// ====== process functions if enabled ======
	// ***** Set Delayed inputs and time elapsed ****
		FB_delIStatus(	IN:= bFcoInputActive,
						PT:= tDelay , 
						Q=> bFcoDelay , 
						ET=> TetInputActive 
					  ); // Generate delayed input status from push button input status
	// ***** Edge triggers *****
		FB_feIStatus(CLK:= Istatus , Q=> bFeStatus ); // generate falling edge pulse on pushbutton input
		FB_reIStatus (Clk := Istatus , Q => bReStatus); // Generate rising edge from push button input signal

END_FUNCTION_BLOCK

// Buttons/Functions/FB_DevPushButton
FUNCTION_BLOCK PUBLIC FB_DevPushButton EXTENDS Fb_DevDigitalInputFunctions
VAR_INPUT
END_VAR
VAR_OUTPUT
END_VAR
VAR
END_VAR

// set device type
IF eDevType = E_Devices.Undefined THEN 
	eDevType := E_Devices.DigitalSensor ;
END_IF

SUPER^();

END_FUNCTION_BLOCK

// Encoders/FunctionBlocks/FB_EncoderBase
FUNCTION_BLOCK PUBLIC FB_EncoderBase
VAR_INPUT
	nCfgUnitsPerPulse	: LREAL := 1	; // Scale factor for output [units/pulse]
	nCfgOffset			: LREAL := 0	; // Offset for output
	
	bIcfInverted		: BOOL	:= FALSE; // Invert output position = standard false  
END_VAR
VAR_OUTPUT
	nOutPosition		: LREAL	:= 0	; // Scaled position output
	nOutRaw				: UDINT := 0	; // Raw output value	 
	nVelocity			: LREAL	:= 0 	; // Velocity [units/sec]
END_VAR
VAR
END_VAR

METHOD PUBLIC FastTask : BOOL
VAR_INPUT
END_VAR
END_METHOD

END_FUNCTION_BLOCK

// Encoders/FunctionBlocks/FB_EncoderInput
FUNCTION_BLOCK FB_EncoderInput EXTENDS FB_EncoderBase
VAR_INPUT
END_VAR
VAR_OUTPUT
END_VAR
VAR
	iEncoderSignal AT%I*: UDINT ;
	
	nScaledValue		: LREAL ; // Only scaled value for internal use
	nValueWithOffset	: LREAL ; // scaled value with added offset
END_VAR

// ====== Scale Output value ======
	nScaledValue := UDINT_TO_LREAL(iEncoderSignal) * nCfgUnitsPerPulse ;

// ====== Invert ======
	IF bIcfInverted THEN 
		nScaledValue := nScaledValue * -1;
	END_IF
	
// ====== Add offset ======= 
	nValueWithOffset := nScaledValue + nCfgOffset ;

// ====== Set Outputs =======
	nOutPosition 	:= nValueWithOffset ;
	nOutRaw			:= iEncoderSignal	;

METHOD PUBLIC FastTask : BOOL
VAR_INPUT
END_VAR
END_METHOD

END_FUNCTION_BLOCK

// HardwareDiagnostics/FB_ELModuleDiag
FUNCTION_BLOCK PUBLIC FB_ELModuleDiag
VAR_INPUT
END_VAR
VAR_OUTPUT
	bError 	:	BOOL ; // Module is in error
	sErrorDiscription : STRING ; // module error discription 
END_VAR
VAR
END_VAR

END_FUNCTION_BLOCK

// Outputs/AnalogOutputs/FB_DevAnalogOutputScaled
FUNCTION_BLOCK FB_DevAnalogOutputScaled EXTENDS FB_DevAnalogOutput
VAR_INPUT
END_VAR
VAR_OUTPUT
END_VAR
VAR
	fGainFactor 	: LREAL:= 32767	;
END_VAR

SUPER^();

METHOD INTERNAL ExecSetFeedback : BOOL
VAR_INPUT
END_VAR
// Set feedback 
fOutputValue := qnHwOut ;
END_METHOD

METHOD INTERNAL ExecSetOutput : BOOL
VAR_INPUT
END_VAR
// Set Output to physical device
IF bEnable OR bCmdManual THEN 
	qnHwOut := LREAL_TO_INT(fCmdValue * fGainFactor) ;
	qnHwOut := LIMIT(nLimitMin, qnHwOut, nLimitMax) ; 
ELSE 
	fCmdValue := 0 ; 
END_IF
END_METHOD

METHOD PUBLIC SetScaling : BOOL 
VAR_INPUT
	fMaxValue	: LREAL ; 		// Maximum input value after scaling, e.g. 100% (mandatory input)  
END_VAR
// calculate gain 
fGainFactor := nLimitMax / fMaxValue ;
END_METHOD

END_FUNCTION_BLOCK

// Sensors/AnalogInput/FunctionBlocks/FB_DevAnalogInAutoCalibrate
FUNCTION_BLOCK PUBLIC FB_DevAnalogInAutoCalibrate EXTENDS FB_DevAnalogInputScaled
VAR_INPUT
END_VAR
VAR_OUTPUT
END_VAR
VAR
END_VAR

SUPER^();

METHOD PUBLIC CmdCalibrateNull : BOOL
VAR_INPUT
END_VAR
// set offset to calibrate to null
nOfset := - inHwInput ;
END_METHOD

METHOD PUBLIC CmdCalilbrateValue : BOOL // calibrate gain factor to actual value (warning calibrate to null before calibrating to value)
VAR_INPUT
	fCalibrationValue	: LREAL ; // Active input value to sensor (calibration setpoint)
END_VAR
// set gain from current value
fGainFactor := INT_TO_LREAL(inHwInput + nOfset) / fCalibrationValue ;
END_METHOD

END_FUNCTION_BLOCK

// Sensors/AnalogInput/FunctionBlocks/FB_DevAnalogInputScaled
FUNCTION_BLOCK PUBLIC FB_DevAnalogInputScaled EXTENDS FB_DevAnalogInput
VAR_INPUT
END_VAR
VAR_OUTPUT
END_VAR
VAR
	fGainFactor 	: LREAL	:= 1	;
	nOfset			: INT	:= 0	;
END_VAR

SUPER^();

METHOD ExecSetFeedback : BOOL
VAR
	nCalibValue	: INT ; 
END_VAR
// Offset 
IF bCmdSimulate THEN 
	nCalibValue := fSimValue + nOfset ;
ELSE
	nCalibValue := inHwInput + nOfset ;
END_IF

fValue := INT_TO_LREAL(nCalibValue) / fGainFactor;
END_METHOD

METHOD PUBLIC SetScaling : BOOL 
VAR_INPUT
	fMaxValue	: LREAL ; 	// Maximum input value after scaling, e.g. 100%, 0 = no scaling (gain = hardware limit / fMaxValue)  
	fOfset		: LREAL ;	// offset value (fvalue = (gain * hwvalue) + fOfset)
END_VAR
// calculate gain 
IF fMaxValue =0 THEN 
	fGainFactor := 1 ;
ELSE 
	fGainFactor := nLimitMax / fMaxValue ;
END_IF

nOfset := LREAL_TO_INT(fOfset * fGainFactor) ;
END_METHOD

END_FUNCTION_BLOCK

// Sensors/AnalogInput/FunctionBlocks/FB_DevHDAnalogInAutoCalibrate
FUNCTION_BLOCK PUBLIC FB_DevHDAnalogInAutoCalibrate EXTENDS FB_DevHDAnalogInputScaled
VAR_INPUT
END_VAR
VAR_OUTPUT
END_VAR
VAR
END_VAR

SUPER^();

METHOD PUBLIC CmdCalibrateNull : BOOL
VAR_INPUT
END_VAR
// set offset to calibrate to null
nOfset := - inHwInput ;
END_METHOD

METHOD PUBLIC CmdCalilbrateValue : BOOL // calibrate gain factor to actual value (warning calibrate to null before calibrating to value)
VAR_INPUT
	fCalibrationValue	: LREAL ; // Active input value to sensor (calibration setpoint)
END_VAR
// set gain from current value
fGainFactor := DINT_TO_LREAL(inHwInput + nOfset) / fCalibrationValue ;
END_METHOD

END_FUNCTION_BLOCK

// Sensors/AnalogInput/FunctionBlocks/FB_DevHDAnalogInputScaled
FUNCTION_BLOCK PUBLIC FB_DevHDAnalogInputScaled EXTENDS FB_DevHDAnalogInput
VAR_INPUT
END_VAR
VAR_OUTPUT
END_VAR
VAR
	fGainFactor 	: LREAL	:= 1	;
	nOfset			: DINT	:= 0	;
END_VAR

SUPER^();

METHOD ExecSetFeedback : BOOL
VAR
	nCalibValue	: DINT ; 
END_VAR
// Offset 
IF bCmdSimulate THEN 
	nCalibValue := fSimValue + nOfset ;
ELSE
	nCalibValue := inHwInput + nOfset ;
END_IF

fValue := DINT_TO_LREAL(nCalibValue) / fGainFactor;
END_METHOD

METHOD PUBLIC SetScaling : BOOL 
VAR_INPUT
	fMaxValue	: LREAL ; 	// Maximum input value after scaling, e.g. 100%, 0 = no scaling (gain = hardware limit / fMaxValue)  
	fOfset		: LREAL ;	// offset value (fvalue = (gain * hwvalue) + fOfset)
END_VAR
// calculate gain 
IF fMaxValue =0 THEN 
	fGainFactor := 1 ;
ELSE 
	fGainFactor := nLimitMax / fMaxValue ;
END_IF

nOfset := LREAL_TO_DINT(fOfset * fGainFactor) ;

SetScaling := TRUE ;
END_METHOD

END_FUNCTION_BLOCK

// Sensors/AnalogInput/FunctionBlocks/FB_DevHDAnalogInput
FUNCTION_BLOCK PUBLIC FB_DevHDAnalogInput EXTENDS FB_DevBase
VAR_INPUT
	bCmdSimulate	: BOOL 	:= FALSE ;// Simulate sensor Input 
	fSimValue		: DINT	:= 0 ;// Simulated sensor state
END_VAR
VAR_OUTPUT
	fValue	: LREAL := 0 ; // Analog input value (LREAL)
END_VAR
VAR
	nLimitMin		: DINT := Utilities_Library.GVL_FixedValues.nDINTMINVALUE	; // Initial value is set to integer minimum value for use with normal def analog inputs 
	nLimitMax 		: DINT := Utilities_Library.GVL_FixedValues.nDINTMAXVALUE 	; // Initial value is set to integer minimum value for use with high def analog inputs
	inHwInput AT%I* : DINT ; // Hardware connection
END_VAR

// Set device type
eDevType := E_Devices.AnalogSensor ;

// Call base function
SUPER^();

// set feedback
ExecSetFeedback();

METHOD ExecSetFeedback : BOOL
VAR_INPUT
END_VAR
IF bCmdSimulate THEN 
	fValue := fSimValue ;
ELSE
	fValue := DINT_TO_LREAL(inHwInput);
END_IF
END_METHOD

END_FUNCTION_BLOCK

// Sensors/FootPedals/FunctionBlocks/FB_EfkaEB301A_FootPedal
FUNCTION_BLOCK PUBLIC FB_EfkaEB301A_FootPedal
VAR_INPUT
	bEnable : BOOL := TRUE ;
END_VAR
VAR_OUTPUT
	ePedalInputStep		: E_FootpedalPos	:= 0 ;
	bRTrigtoReverse1 	: BOOL := FALSE ; // rising edge trigger when pedal moves from 0 to -1 or Idle to reverse 1 
	bRTrigtoReverse2 	: BOOL := FALSE ; // rising edge trigger when pedal moves from 1 to -2 or reverse 1 to reverse 2 
	bRTrigtoForward1 	: BOOL := FALSE ; // rising edge trigger when pedal moves from 0 to 1 or idle to forward 1 
	bRTrigtoForward2 	: BOOL := FALSE ; // rising edge trigger when pedal moves from 0 to 1 or forward to forward 2 
END_VAR
VAR
	// ===== greycode switches from footpedal =====
	I_GreyCodeA AT%I* : BOOL	; // Greycode input a from foot pedal 
	I_GreyCodeB AT%I* : BOOL	; // Greycode input a from foot pedal 
	I_GreyCodeC AT%I* : BOOL	; // Greycode input a from foot pedal 
	I_GreyCodeD AT%I* : BOOL	; // Greycode input a from foot pedal 
	nGreyCodetotal	: BYTE ; // all greycode switches combined
	// ==== decimal value =====
	ePreviousPedalInput	: E_FootpedalPos	:= 0 ;
END_VAR

// ===== Read input from pedal =====
ACT_ConvertGreycode();

// ===== Create edge flanks for functions =====
ACT_CreateEdges();

ACTION ACT_ConvertGreycode:
// ===== Combine greycode sensors =====
nGreyCodetotal.0 := I_GreyCodeA ;
nGreyCodetotal.1 := I_GreyCodeB ;
nGreyCodetotal.2 := I_GreyCodeB ;
nGreyCodetotal.3 := I_GreyCodeC ;

// ==== Convert greycode decimal to speed steps =====
// this only makes sense in EFKA world but anyway let's convert it to our own sense
CASE nGreyCodetotal OF 
	12: ePedalInputStep := E_FootpedalPos.eReverse1	;
	14: ePedalInputStep := E_FootpedalPos.eReverse2	;
	15: ePedalInputStep := E_FootpedalPos.eIdle		;
	13: ePedalInputStep := E_FootpedalPos.eForward1	;
	09: ePedalInputStep := E_FootpedalPos.eForward2	;
 	08: ePedalInputStep := E_FootpedalPos.eForward3	;
	10: ePedalInputStep := E_FootpedalPos.eForward4	;
	11: ePedalInputStep := E_FootpedalPos.eForward5	;
	03:	ePedalInputStep := E_FootpedalPos.eForward6	;
	02:	ePedalInputStep := E_FootpedalPos.eForward7	;
	00: ePedalInputStep := E_FootpedalPos.eForward8	;
	01: ePedalInputStep := E_FootpedalPos.eForward9	;
	05: ePedalInputStep := E_FootpedalPos.eForward10	;
	04: ePedalInputStep := E_FootpedalPos.eForward11	;
	06: ePedalInputStep := E_FootpedalPos.eForward12 	;
	07: ePedalInputStep := E_FootpedalPos.eForward13	;
	ELSE
		ePedalInputStep := E_FootpedalPos.eFalse 		;
END_CASE
END_ACTION

ACTION ACT_CreateEdges:
// ===== create edges on which functions can be triggerd =====
CASE ePedalInputStep OF
	E_FootpedalPos.eReverse2:
		bRTrigtoReverse2 := ePreviousPedalInput = E_FootpedalPos.eReverse1 ;
	E_FootpedalPos.eReverse1:
		bRTrigtoReverse1 := ePreviousPedalInput = E_FootpedalPos.eIdle ;
	E_FootpedalPos.eForward1:
		bRTrigtoForward1 := ePreviousPedalInput = E_FootpedalPos.eIdle ;
	E_FootpedalPos.eForward2: 
		bRTrigtoForward2 := ePreviousPedalInput = E_FootpedalPos.eForward1 ; 
END_CASE 

// write previous pedal input 
ePreviousPedalInput := ePedalInputStep ;
END_ACTION

END_FUNCTION_BLOCK

// Sensors/ModuleSpecific/EL3556_Loadcell/Fb_DevEL3356_LoadCell
FUNCTION_BLOCK PUBLIC Fb_DevEL3356_LoadCell EXTENDS FB_DevHDAnalogInAutoCalibrate
VAR_INPUT
	tCalibrationDelay	: TIME := T#2S ; // Time for which the load neads to before calibration is done (default T#2s) 
END_VAR
VAR_OUTPUT
	bMeasurementError	: BOOL 		; // Measurement or component error is active
	sErroDiscription 	: STRING 	; // 
END_VAR
VAR
	ibOverrange				AT%I*	: BOOL ; // overrange status indication
	ibDataInvalid			AT%I*	: BOOL ; // Data is invalid
	ibError					AT%I*	: BOOL ; // Module is in error state
	ibCalibrationinProgress	AT%I*	: BOOL ; // automatic calibration is in progress
	ibSteadyState			AT%I*	: BOOL ; // Module is in steady state
	ibSyncError				AT%I*	: BOOL ; // Module sync error
	
	tonSteadyState	: TON ; // steady state delay for calibration
END_VAR

ACTION CheckELSignalState:
// Set error device measurement error bit
bMeasurementError := FALSE ;

IF ibOverrange THEN 
	bMeasurementError 	S= TRUE;
 	sErroDiscription	:= 'Load exceeds maximum range ';
ELSIF ibDataInvalid THEN
	bMeasurementError 	S= TRUE;
	sErroDiscription	:= 'Incorrect date from device';
ELSIF ibError THEN
	bMeasurementError 	S= TRUE;
	sErroDiscription	:= 'Module general error';
ELSIF ibCalibrationinProgress THEN
	bMeasurementError 	S= TRUE;
	sErroDiscription	:= 'Calibration session in progress';
ELSIF ibSyncError THEN
	bMeasurementError 	S= TRUE;
	sErroDiscription	:= 'Module ethercat sync error';	
END_IF
END_ACTION

METHOD PUBLIC CmdCalibrateNull : BOOL
VAR_INPUT
END_VAR
tonSteadyState(IN := ibSteadyState, PT := tCalibrationDelay);

// set offset to calibrate to null
IF tonSteadyState.Q THEN 
	nOfset := - inHwInput ;
END_IF
END_METHOD

METHOD PUBLIC CmdCalilbrateValue : BOOL // calibrate gain factor to actual value (warning calibrate to null before calibrating to value)
VAR_INPUT
	fCalibrationValue	: LREAL ; // Active input value to sensor [N]
END_VAR
tonSteadyState(IN := ibSteadyState, PT := tCalibrationDelay);

// set gain from current value
IF tonSteadyState.Q THEN 
	fGainFactor := DINT_TO_LREAL(inHwInput + nOfset) / fCalibrationValue ; 
END_IF
END_METHOD

END_FUNCTION_BLOCK
